FUNCTION_BLOCK Motor_VS (* CAT Function Block Type *)
  (* Standard: 61499-2 *)
  (* Version 0.0, 6/2/2026, Schneider Electric, template *)
  PACKAGE SE.Nereda;
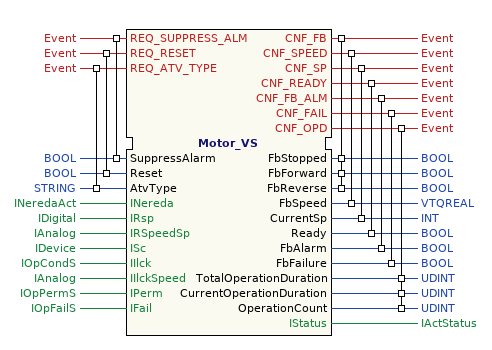
  EVENT_INPUT
    REQ_SUPPRESS_ALM WITH SuppressAlarm; (* Request to update the alarm suppress status *)
    REQ_RESET WITH Reset; (* Request to reset the device *)
    REQ_ATV_TYPE WITH AtvType;
  END_EVENT
  EVENT_OUTPUT
    CNF_FB WITH FbStopped, FbForward, FbReverse; (* Execution of confirmed state *)
    CNF_SPEED WITH FbSpeed; (* Execution of confirmed state *)
    CNF_SP WITH CurrentSp; (* Execution of confirmation current setpoint *)
    CNF_READY WITH Ready; (* Execution of Ready status *)
    CNF_FB_ALM WITH FbAlarm; (* Execution of confirmation  Fb alarm *)
    CNF_FAIL WITH FbFailure; (* Execution of confirmation  failure *)
    CNF_OPD WITH TotalOperationDuration, CurrentOperationDuration, OperationCount; (* Execution confirmation of operation durations *)
  END_EVENT
  VAR_INPUT
    SuppressAlarm : BOOL; (* 1 = Suppress alarm in HMI *)
    Reset : BOOL; (* 1 = Reset device failure *)
    AtvType : STRING;
  END_VAR
  VAR_OUTPUT
    FbStopped : BOOL; (* 1 = Stopped *)
    FbForward : BOOL; (* 1 = Running *)
    FbReverse : BOOL; (* 1 = Running *)
    FbSpeed : VTQREAL; (* Value from the hardware module *)
    CurrentSp : INT; (* Current output value considering permissive conditions *)
    Ready : BOOL; (* 1 = Device is ready to run *)
    FbAlarm : BOOL; (* 1 = Feedback failure alarm is active *)
    FbFailure : BOOL; (* 1 = Fail active *)
    TotalOperationDuration : UDINT; (* Total operation duration in minutes *)
    CurrentOperationDuration : UDINT; (* Current operational duration in minutes *)
    OperationCount : UDINT; (* Total operations count *)
  END_VAR
  SOCKETS
    INereda : INeredaAct;
  END_SOCKETS
  SOCKETS
    IRsp : IDigital; (* Program remote setpoint interface adapter *)
    IRSpeedSp : IAnalog; (* Program remote speed setpoint interface adpter, Controls the block when owner is in program local. *)
    ISc : IDevice; (* Sequence control Interface adapter. Controls the block when owner is in program local *)
    IIlck : IOpCondS; (* Condition summary chain input from upstream blocks *)
    IIlckSpeed : IAnalog; (* Speed setpoint to be considered if interlock condition is active *)
    IPerm : IOpPermS; (* Permission condition summary chain input from permCondItem blocks *)
    IFail : IOpFailS; (* Fail condition summary chain input from failCondItem blocks *)
  END_SOCKETS
  PLUGS
    IStatus : IActStatus;
  END_PLUGS
  (* 01 - FUNCTIONNAL INPUT INTERFACE *)
  (* 00 - INITIALIZATION *)
  (* 05 - LOGIC *)
  (* 06 - HMI INTERFACE *)
  (* 04 - CHILDREN *)
  (* 03 - FIELD INTERFACE *)
  (* 02 - FUNCTIONNAL OUTPUT INTERFACE *)
  (* 07- Input Hardware Interface *)
  (* 08- Output Hardware Interface *)
  (* 09- Local Panel *)
  (* Maintenance *)
  (* Fb Stop *)
  (* Interlock *)
  (* Mode *)
  (* Permissive *)
  (* 4A - TYPICALS *)
  (* Craeted By Nouriddin OUECHEN *)
  (* Failure *)
  (* Sequence Control *)
  (* Service Connection *)
  (* Reset *)
  (* FbRunning *)
  (* SetPoint *)
  (* Simulation (To be Removed) *)
  (* 07- ±OTOR VS ALARM *)
  (* Comment When `SafetySwitchOff = TRUE`, it means that the safety switch is **OFF**. *)
  FBS
    IThis : Motor_VS_HMI(QI := TRUE);
    INIT : plcStart(Prio := 35, Delay := T#0ms);
    extControlled : dISignal(Name := '$${PATH}DIn'); {SET_ATTRIBUTE(Configuration.Component.HideUnusedPorts, )}
    LocalPanel : FieldSignals;
    maintenance : DevMnt; {SET_ATTRIBUTE(Configuration.Component.HideUnusedPorts, )}
    NotRevFwd : NOT_425622A9A4AC6C60; {SET_ATTRIBUTE(Configuration.GenericFBType.InterfaceParams, Runtime.Standard#CNT:=2;OUT${CNT$}:BOOL,BOOL)}
    interlock : IlckCondSum; {SET_ATTRIBUTE(Configuration.Component.HideUnusedPorts, )}
    failure : FailCondSum; {SET_ATTRIBUTE(Configuration.Component.HideUnusedPorts, )}
    DriveFailure : failCondItem(CondCause := Active1); {SET_ATTRIBUTE(Configuration.Component.HideUnusedPorts, )}
    AtvFailure : SELECT_81F91C08E00C8B28(IN1 := FALSE); {SET_ATTRIBUTE(Configuration.GenericFBType.InterfaceParams, Runtime.Standard#CNT:=2;SELECT:BOOL;IN${CNT$}:BOOL)}
    ElectricCircuitFailure : failCondItem(CondCause := Active1); {SET_ATTRIBUTE(Configuration.Component.HideUnusedPorts, )}
    FrequencyInverterFailure : failCondItem(CondCause := Active1); {SET_ATTRIBUTE(Configuration.Component.HideUnusedPorts, )}
    PowerFailure : failCondItem(CondCause := Active1); {SET_ATTRIBUTE(Configuration.Component.HideUnusedPorts, )}
    CurrOwner : CurrOwnerDecode;
    State : ActState(pin_DD241BABAE81E6FD := Motor);
    NoPowerFb : NOT_42C76073DCEB1A7A; {SET_ATTRIBUTE(Configuration.GenericFBType.InterfaceParams, Runtime.Standard#CNT:=1;OUT${CNT$}:BOOL)}
    permissive : PermCondSum; {SET_ATTRIBUTE(Configuration.Component.HideUnusedPorts, )}
    BaseVs : MotorVsBase;
    interlockMotVs : IlckMotVs;
    fbFwd : dISignal(Name := '$${PATH}DIn'); {SET_ATTRIBUTE(Configuration.Component.HideUnusedPorts, )}
    fbRev : dISignal(Name := '$${PATH}DIn'); {SET_ATTRIBUTE(Configuration.Component.HideUnusedPorts, )}
    fbSpeed : aISignal(Name := '$${PATH}AIn'); (* (Minimum Value  = 0.0, Maximum Value = 100.0) *) {SET_ATTRIBUTE(Configuration.Component.HideUnusedPorts, )}
    FbStop : AND_88A3DD8EC65DD11C; {SET_ATTRIBUTE(Configuration.GenericFBType.InterfaceParams, Runtime.Standard#CNT:=2;OUT:BOOL)}
    serviceManager : MotorVsServiceManager; {SET_ATTRIBUTE(Configuration.Component.HideUnusedPorts, )}
    cmdFwd : dOSignal(Name := '$${PATH}DOut'); {SET_ATTRIBUTE(Configuration.Component.HideUnusedPorts, )}
    cmdSpeed : aOSignal(Name := '$${PATH}AOut'); {SET_ATTRIBUTE(Configuration.Component.HideUnusedPorts, )}
    cmdRev : dOSignal(Name := '$${PATH}DOut'); {SET_ATTRIBUTE(Configuration.Component.HideUnusedPorts, )}
    ResetCmd : OR_169B00D031196E7C4; {SET_ATTRIBUTE(Configuration.GenericFBType.InterfaceParams, Runtime.Standard#CNT:=4;OUT:BOOL)}
    FbRunning : OR_88A3DD8EC65DD11C; {SET_ATTRIBUTE(Configuration.GenericFBType.InterfaceParams, Runtime.Standard#CNT:=2;OUT:BOOL)}
    ISc1ISc2 : mergeIDevice;
    Sp : IDeviceEncode;
    IScISeqData : IScISecData;
    TRIP : failCondItem(CondCause := Active1); {SET_ATTRIBUTE(Configuration.Component.HideUnusedPorts, )}
    MoistureDetectionPumpMS : failCondItem(CondCause := Active1); {SET_ATTRIBUTE(Configuration.Component.HideUnusedPorts, )}
    Reset_Init : DS_SELECTX_2536758B411A6CE51(DI1_1 := TRUE, DI2_1 := FALSE); {SET_ATTRIBUTE(Configuration.GenericFBType.InterfaceParams, Runtime.Standard#CNTX:=2;CNTY:=1;DI${CNTX,_,CNTY$}:BOOL)}
    NoNeedReset : E_PERMIT;
    NotNeedReset : NOT_42C76073DCEB1A7A; {SET_ATTRIBUTE(Configuration.GenericFBType.InterfaceParams, Runtime.Standard#CNT:=1;OUT${CNT$}:BOOL)}
    SpeedSp : SpeedSp;
    SafetySwitchOff : ilckCondItem(CondCause := Active1);
    SafetySwitch : NOT_42C76073DCEB1A7A; {SET_ATTRIBUTE(Configuration.GenericFBType.InterfaceParams, Runtime.Standard#CNT:=1;OUT${CNT$}:BOOL)}
    AllFailures : OR_1147623A96AA66A8; {SET_ATTRIBUTE(Configuration.GenericFBType.InterfaceParams, Runtime.Standard#CNT:=7;OUT:BOOL)}
    AlarmDriveFailure : ALARM_BIT(ACKTYPE_1 := 2, ACTIVE := TRUE, TYPE := 1);
    AlarmTRIP : ALARM_BIT(ACKTYPE_1 := 2, TYPE := 1, ACTIVE := TRUE);
    AlarmElectricCircuitFailure : ALARM_BIT(ACKTYPE_1 := 2, ACTIVE := TRUE, TYPE := 1);
    AlarmFrequencyInverterFailure : ALARM_BIT(ACKTYPE_1 := 2, ACTIVE := TRUE, TYPE := 1);
    AlarmPowerFailure : ALARM_BIT(ACKTYPE_1 := 2, ACTIVE := TRUE, TYPE := 1);
    AlarmMoistureDetectionPumpMS : ALARM_BIT(ACKTYPE_1 := 2, ACTIVE := TRUE, TYPE := 1);
    MotorVsFailuresAlarms : MotVsFailures;
    MUL1 : MUL_1329C2AB45109BAAB(IN2 := 0.6); {SET_ATTRIBUTE(Configuration.GenericFBType.InterfaceParams, Runtime.Standard#CNT:=2;IN${CNT$}:REAL)}
    SYMLINKMULTIVARSRC1 : SYMLINKMULTIVARSRC_5A03F112CD5D470(QI := TRUE, NAME1 := '$${PATH}cmdFrequency'); {SET_ATTRIBUTE(Configuration.GenericFBType.InterfaceParams, Runtime.System#I:=1;VALUE${I$}:INT)}
    REAL2INT1 : REAL2INT;
    SYMLINKMULTIVARSRC2 : SYMLINKMULTIVARSRC_5A03F112CD5D470(QI := TRUE, NAME1 := '$${PATH}cmdSpeedINT'); {SET_ATTRIBUTE(Configuration.GenericFBType.InterfaceParams, Runtime.System#I:=1;VALUE${I$}:INT)}
    SpeedRawOut : speedToRawInt(pin_EEBD45F5182DE80D := 100.0);
    FbSpeedAdapter : speedFbAdapter(pin_919EBDC14EE69C57 := 100.0);
    fbSpeedINT : SYMLINKMULTIVARDST_5A03F112CD5D470(QI := TRUE, NAME1 := '$${PATH}fbSpeedINT'); {SET_ATTRIBUTE(Configuration.GenericFBType.InterfaceParams, Runtime.System#I:=1;VALUE${I$}:INT)}
  END_FBS
  EVENT_CONNECTIONS
    extControlled.CNF TO BaseVs.REQ_EXT_CTL;
    failure.COND_IND TO BaseVs.REQ_FAIL;
    REQ_SUPPRESS_ALM TO BaseVs.REQ_SUPPRESS_ALM;
    BaseVs.CNF_FB_STS TO CNF_FB;
    BaseVs.CNF_FB_ALM TO CNF_FB_ALM;
    State.7E9F7DF9BBDC513D TO CNF_FAIL;
    NoPowerFb.CNF TO DriveFailure.REQ;
    NoPowerFb.CNF TO ElectricCircuitFailure.REQ;
    NoPowerFb.CNF TO FrequencyInverterFailure.REQ;
    NoPowerFb.CNF TO PowerFailure.REQ;
    permissive.PERM_IND TO BaseVs.REQ_PERM;
    AtvFailure.CNF TO NoPowerFb.REQ;
    FbSpeedAdapter.DCDCAD18DFD61DDE TO BaseVs.REQ_FB_SPEED;
    fbFwd.CNF TO NotRevFwd.REQ;
    fbRev.CNF TO NotRevFwd.REQ;
    FbStop.CNF TO BaseVs.REQ_FB;
    NotRevFwd.CNF TO FbStop.REQ;
    BaseVs.CNF_OUT TO cmdFwd.REQ;
    BaseVs.CNF_OUT TO cmdRev.REQ;
    BaseVs.CNF_SPEED_OUT TO cmdSpeed.REQ;
    FbSpeedAdapter.DCDCAD18DFD61DDE TO CNF_SPEED;
    BaseVs.CNF_SP TO CNF_SP;
    maintenance.CNF_OPD TO CNF_OPD;
    BaseVs.CNF_FB_STS TO FbRunning.REQ;
    NoPowerFb.CNF TO TRIP.REQ;
    NoPowerFb.CNF TO MoistureDetectionPumpMS.REQ;
    REQ_RESET TO ResetCmd.REQ;
    ResetCmd.CNF TO BaseVs.REQ_RESET;
    Reset_Init.IND TO ResetCmd.REQ;
    NotNeedReset.CNF TO NoNeedReset.EI;
    BaseVs.CNF_NEED_RESET TO NotNeedReset.REQ;
    NoNeedReset.EO TO Reset_Init.REQ2;
    LocalPanel.08EBB16DA2AE2E53 TO AtvFailure.REQ;
    CurrOwner.7B1DE71047870DF3 TO State.503DFB34A9D9F842;
    State.B9B326A02DDC85D5 TO AlarmDriveFailure.INIT;
    State.B9B326A02DDC85D5 TO NotRevFwd.REQ;
    State.B9B326A02DDC85D5 TO IScISeqData.68E777F8FBF99C3F;
    State.B9B326A02DDC85D5 TO Sp.6454C45AB89C818D;
    State.B9B326A02DDC85D5 TO Reset_Init.REQ1;
    State.3E2F994B40CA5D8A TO CNF_READY;
    State.3E2F994B40CA5D8A TO INereda.CC753684FA882790;
    State.3E2F994B40CA5D8A TO IStatus.14377629A1F197A9;
    REQ_ATV_TYPE TO LocalPanel.62FE49324B71C4B0;
    FbRunning.CNF TO INereda.9CD053F8408797ED;
    FbSpeedAdapter.DCDCAD18DFD61DDE TO INereda.F846995A4121D865;
    BaseVs.CNF_FB_ALM TO INereda.C79FD2A34D0395C5;
    State.7E9F7DF9BBDC513D TO INereda.476AAA40EB7AA926;
    maintenance.CNF_OPD TO INereda.2DA8AEC15204E92D;
    INereda.0F1CDF9A9B4A227A TO BaseVs.REQ_SP;
    INereda.0F1CDF9A9B4A227A TO Sp.7A6C1C05B7ACA4D3;
    INereda.0F1CDF9A9B4A227A TO SpeedSp.3B62B1C54EE8482F;
    INereda.1E00729184986247 TO SpeedSp.3B62B1C54EE8482F;
    INereda.37BBC1F841739733 TO Sp.8DD7A09A6565B7F3;
    INereda.37BBC1F841739733 TO ResetCmd.REQ;
    SpeedSp.CE921AF394A1453E TO Sp.51FC99EF6C596181;
    BaseVs.CNF_MODE TO interlockMotVs.BB07CE5CA3A90E8C;
    BaseVs.CNF_OWNER TO interlockMotVs.47593EB5799F5830;
    interlockMotVs.1ACB26BE744F37A1 TO BaseVs.REQ_ILCK;
    FbRunning.CNF TO IStatus.14377629A1F197A9;
    FbSpeedAdapter.DCDCAD18DFD61DDE TO IStatus.03F1F1C982EE8DD5;
    SafetySwitch.CNF TO SafetySwitchOff.REQ;
    LocalPanel.08EBB16DA2AE2E53 TO SafetySwitch.REQ;
    LocalPanel.08EBB16DA2AE2E53 TO AllFailures.REQ;
    BaseVs.CNF_SP TO AllFailures.REQ;
    BaseVs.CNF_FB_STS TO AllFailures.REQ;
    BaseVs.CNF_OWNER TO AllFailures.REQ;
    BaseVs.CNF_READY TO AllFailures.REQ;
    BaseVs.CNF_MODE TO AllFailures.REQ;
    interlockMotVs.1ACB26BE744F37A1 TO AllFailures.REQ;
    BaseVs.CNF_FAIL TO AllFailures.REQ;
    AllFailures.CNF TO CurrOwner.3D8B91432EBB5812;
    NoPowerFb.CNF TO AllFailures.REQ;
    BaseVs.CNF_NEED_RESET TO AllFailures.REQ;
    AlarmPowerFailure.INITO TO AlarmTRIP.INIT;
    AlarmDriveFailure.INITO TO AlarmElectricCircuitFailure.INIT;
    AlarmElectricCircuitFailure.INITO TO AlarmFrequencyInverterFailure.INIT;
    AlarmDriveFailure.CNF_INITDATA TO AlarmDriveFailure.REQ;
    MotorVsFailuresAlarms.C14C3E40270A0244 TO AlarmDriveFailure.REQ_INITDATA;
    MotorVsFailuresAlarms.C14C3E40270A0244 TO AlarmTRIP.REQ_INITDATA;
    AlarmTRIP.CNF_INITDATA TO AlarmTRIP.REQ;
    AlarmDriveFailure.CNF_INITDATA TO AlarmDriveFailure.ACTIVATE;
    AlarmTRIP.CNF_INITDATA TO AlarmTRIP.ACTIVATE;
    AlarmFrequencyInverterFailure.INITO TO AlarmPowerFailure.INIT;
    MotorVsFailuresAlarms.C14C3E40270A0244 TO AlarmElectricCircuitFailure.REQ_INITDATA;
    MotorVsFailuresAlarms.C14C3E40270A0244 TO AlarmFrequencyInverterFailure.REQ_INITDATA;
    MotorVsFailuresAlarms.C14C3E40270A0244 TO AlarmPowerFailure.REQ_INITDATA;
    AlarmElectricCircuitFailure.CNF_INITDATA TO AlarmElectricCircuitFailure.ACTIVATE;
    AlarmElectricCircuitFailure.CNF_INITDATA TO AlarmElectricCircuitFailure.REQ;
    AlarmFrequencyInverterFailure.CNF_INITDATA TO AlarmFrequencyInverterFailure.ACTIVATE;
    AlarmFrequencyInverterFailure.CNF_INITDATA TO AlarmFrequencyInverterFailure.REQ;
    AlarmPowerFailure.CNF_INITDATA TO AlarmPowerFailure.ACTIVATE;
    AlarmPowerFailure.CNF_INITDATA TO AlarmPowerFailure.REQ;
    MotorVsFailuresAlarms.C14C3E40270A0244 TO AlarmMoistureDetectionPumpMS.REQ_INITDATA;
    AlarmMoistureDetectionPumpMS.CNF_INITDATA TO AlarmMoistureDetectionPumpMS.ACTIVATE;
    AlarmMoistureDetectionPumpMS.CNF_INITDATA TO AlarmMoistureDetectionPumpMS.REQ;
    AlarmTRIP.INITO TO AlarmMoistureDetectionPumpMS.INIT;
    NoPowerFb.CNF TO AlarmDriveFailure.REQ;
    NoPowerFb.CNF TO AlarmElectricCircuitFailure.REQ;
    NoPowerFb.CNF TO AlarmFrequencyInverterFailure.REQ;
    NoPowerFb.CNF TO AlarmPowerFailure.REQ;
    NoPowerFb.CNF TO AlarmTRIP.REQ;
    NoPowerFb.CNF TO AlarmMoistureDetectionPumpMS.REQ;
    AlarmMoistureDetectionPumpMS.INITO TO MotorVsFailuresAlarms.5D68F3F24BC03060;
    AlarmDriveFailure.IND_1 TO MotorVsFailuresAlarms.BB7D0193D5CDB632;
    AlarmElectricCircuitFailure.IND_1 TO MotorVsFailuresAlarms.BB7D0193D5CDB632;
    AlarmFrequencyInverterFailure.IND_1 TO MotorVsFailuresAlarms.BB7D0193D5CDB632;
    AlarmPowerFailure.IND_1 TO MotorVsFailuresAlarms.BB7D0193D5CDB632;
    AlarmTRIP.IND_1 TO MotorVsFailuresAlarms.BB7D0193D5CDB632;
    AlarmMoistureDetectionPumpMS.IND_1 TO MotorVsFailuresAlarms.BB7D0193D5CDB632;
    INIT.FIRST_INIT TO IThis.5D65C7F23F6CCFDB;
    INIT.REDO_INIT TO IThis.5D65C7F23F6CCFDB;
    State.B9B326A02DDC85D5 TO IThis.D29F1FADF6E57358;
    LocalPanel.08EBB16DA2AE2E53 TO IThis.438D25703EEFF814;
    BaseVs.CNF_SPEED_SP TO IThis.0316FFC0BDC899BE;
    FbSpeedAdapter.DCDCAD18DFD61DDE TO IThis.0316FFC0BDC899BE;
    BaseVs.CNF_NEED_RESET TO IThis.05E2BC0E0C273F8B;
    State.7E9F7DF9BBDC513D TO IThis.A2D93536FF9B406B;
    fbFwd.CNF TO IThis.C9F8920D38B4A811;
    IThis.141F2765F0199247 TO State.747A80A26976E9BA;
    IThis.EDABC861E1C71398 TO AtvFailure.REQ;
    IThis.6535878B6880E95C TO ResetCmd.REQ;
    IThis.52FEB725938026A3 TO BaseVs.REQ_SPEED_SP;
    BaseVs.CNF_SPEED_OUT TO MUL1.REQ;
    MUL1.CNF TO REAL2INT1.DD5870AA881150BB;
    MotorVsFailuresAlarms.C14C3E40270A0244 TO fbSpeedINT.INIT;
    REAL2INT1.6FC99A5BD1C38561 TO SYMLINKMULTIVARSRC1.REQ;
    SYMLINKMULTIVARSRC1.INITO TO INIT.ACK_FIRST;
    BaseVs.CNF_SPEED_OUT TO SpeedRawOut.45891852F5D66F4B;
    SpeedRawOut.73091BCABFCCFCB6 TO SYMLINKMULTIVARSRC2.REQ;
    SYMLINKMULTIVARSRC2.INITO TO SYMLINKMULTIVARSRC1.INIT;
    fbSpeed.CNF TO FbSpeedAdapter.23AEC014E6AA5B8A;
    fbSpeedINT.CNF TO FbSpeedAdapter.D15EB431906F2F27;
    fbSpeedINT.INITO TO SYMLINKMULTIVARSRC2.INIT;
  END_CONNECTIONS
  DATA_CONNECTIONS
    extControlled.Out TO BaseVs.ExternalControlled;
    fbFwd.Out TO BaseVs.FbFwd;
    failure.State TO BaseVs.Fail;
    SuppressAlarm TO BaseVs.SuppressAlarm;
    BaseVs.FbStopped TO FbStopped;
    BaseVs.FbFwdRunning TO FbForward;
    BaseVs.FbAlarm TO FbAlarm;
    State.8CCAFBE354ECA569 TO FbFailure;
    AtvFailure.OUT TO DriveFailure.CondSignal;
    NoPowerFb.OUT1 TO PowerFailure.CondSignal;
    permissive.PermPassive TO BaseVs.PermStop;
    permissive.PermActive1 TO BaseVs.PermFwd;
    fbRev.Out TO BaseVs.FbRev;
    FbSpeedAdapter.02242968B1987D9E TO BaseVs.FbSpeed;
    fbFwd.Out TO NotRevFwd.IN1;
    FbStop.OUT TO BaseVs.FbStop;
    fbRev.Out TO NotRevFwd.IN2;
    NotRevFwd.OUT1 TO FbStop.IN1;
    NotRevFwd.OUT2 TO FbStop.IN2;
    permissive.PermActive2 TO BaseVs.PermRev;
    BaseVs.OutFwd TO cmdFwd.Signal;
    BaseVs.OutRev TO cmdRev.Signal;
    BaseVs.OutSpeed TO cmdSpeed.Signal;
    FbSpeedAdapter.02242968B1987D9E TO FbSpeed;
    BaseVs.FbRevRunning TO FbReverse;
    BaseVs.CurrentSp TO CurrentSp;
    maintenance.TotalOperationDuration TO TotalOperationDuration;
    maintenance.CurrentOperationDuration TO CurrentOperationDuration;
    maintenance.OperationCount TO OperationCount;
    BaseVs.FbFwdRunning TO FbRunning.IN1;
    BaseVs.FbRevRunning TO FbRunning.IN2;
    Reset TO ResetCmd.IN1;
    ResetCmd.OUT TO BaseVs.Reset;
    Reset_Init.OUT1 TO ResetCmd.IN4;
    NotNeedReset.OUT1 TO NoNeedReset.PERMIT;
    BaseVs.NeedReset TO NotNeedReset.IN1;
    LocalPanel.9DA3D6735086B77A TO ElectricCircuitFailure.CondSignal;
    LocalPanel.B021B183D08305E2 TO FrequencyInverterFailure.CondSignal;
    LocalPanel.DA445F1C2864A153 TO State.C70237F918BB93F6;
    LocalPanel.B46B24B64003C584 TO NoPowerFb.IN1;
    LocalPanel.B46B24B64003C584 TO State.655DE7D6E2CF8FB8;
    LocalPanel.61B515FEF739774D TO AtvFailure.IN2;
    LocalPanel.4379EE93CED9D91D TO TRIP.CondSignal;
    LocalPanel.5EFEAD483C25BA7B TO MoistureDetectionPumpMS.CondSignal;
    CurrOwner.CEBE936F1EA616DB TO State.E90E39DE4A80ABDE;
    CurrOwner.1FF13EB8D921FC26 TO State.3885B231A80F7FFF;
    BaseVs.CurrentOwner TO CurrOwner.B2DAC483AB345195;
    State.4E509FA35DBACB85 TO Ready;
    State.4E509FA35DBACB85 TO INereda.8A8A07EFCDA1443C;
    State.4E509FA35DBACB85 TO IStatus.9E0B44559326BEAF;
    BaseVs.CurrentSp TO State.52C3EF6D9E750127;
    BaseVs.FbStatus TO State.8E076A9FED13120E;
    BaseVs.Ready TO State.1C9201C719ABF50B;
    BaseVs.Simulation TO State.7A0BDA68B634A263;
    BaseVs.FbOverride TO State.DD66F5DCF7F6FB1D;
    interlockMotVs.74F62D32B8AB17CB TO State.9A204E382C1350DC;
    AtvType TO LocalPanel.62A70FF94078EC4D;
    BaseVs.FbStopped TO INereda.D83B5BDEFA4D797C;
    FbRunning.OUT TO INereda.B762734C094A7162;
    BaseVs.FbFwdRunning TO INereda.13E1B1B6EE0F07DB;
    BaseVs.FbRevRunning TO INereda.3011FF733C667A56;
    FbSpeedAdapter.02242968B1987D9E TO INereda.790C5C3BA88E0AF5;
    BaseVs.FbAlarm TO INereda.BDD69968F2D82EAF;
    State.8CCAFBE354ECA569 TO INereda.6EEAF63EEE6021B6;
    maintenance.TotalOperationDuration TO INereda.C7F638DBF6B860D2;
    maintenance.CurrentOperationDuration TO INereda.9224E22E0E82A2D7;
    maintenance.OperationCount TO INereda.10624535249F94F3;
    INereda.710D7FC54EE3F35A TO BaseVs.Sp;
    INereda.710D7FC54EE3F35A TO Sp.64F0A65D5B10944D;
    INereda.710D7FC54EE3F35A TO SpeedSp.28B1E385E2B35AAE;
    INereda.1BC103921BBFDA0B TO SpeedSp.79740CC6CE911CBD;
    INereda.EA28053F07575F36 TO Sp.48AF5FD15A286274;
    INereda.EA28053F07575F36 TO ResetCmd.IN3;
    SpeedSp.335EA17E377251F8 TO Sp.35DB549676DB86DA;
    BaseVs.Maintenance TO interlockMotVs.3100FF95313D2E79;
    BaseVs.CurrentOwner TO interlockMotVs.B24A2EB6CD7D5206;
    interlockMotVs.5B70B8A759686CBA TO BaseVs.IlckPos;
    interlockMotVs.5CCAAE9E9D3EC477 TO BaseVs.IlckType;
    interlockMotVs.7BFBF177262F6463 TO BaseVs.IlckSpeed;
    BaseVs.FbStopped TO IStatus.227987A2F0C6A825;
    FbRunning.OUT TO IStatus.D41A46B14EF7208D;
    FbSpeedAdapter.02242968B1987D9E TO IStatus.B9E42D72CEF16844;
    SafetySwitch.OUT1 TO SafetySwitchOff.CondSignal;
    LocalPanel.9F4FA80000721942 TO SafetySwitch.IN1;
    interlockMotVs.74F62D32B8AB17CB TO BaseVs.IlckCond;
    BaseVs.FbAlarm TO State.F37ACDE435F84908;
    BaseVs.FailStatus TO AllFailures.IN1;
    AtvFailure.OUT TO AllFailures.IN2;
    LocalPanel.9DA3D6735086B77A TO AllFailures.IN3;
    LocalPanel.B021B183D08305E2 TO AllFailures.IN4;
    NoPowerFb.OUT1 TO AllFailures.IN5;
    LocalPanel.4379EE93CED9D91D TO AllFailures.IN6;
    LocalPanel.5EFEAD483C25BA7B TO AllFailures.IN7;
    AllFailures.OUT TO State.94E3C396E1CCD1C0;
    BaseVs.NeedReset TO State.3ED730632EF45559;
    AtvFailure.OUT TO AlarmDriveFailure.INP;
    LocalPanel.9DA3D6735086B77A TO AlarmElectricCircuitFailure.INP;
    LocalPanel.B021B183D08305E2 TO AlarmFrequencyInverterFailure.INP;
    NoPowerFb.OUT1 TO AlarmPowerFailure.INP;
    LocalPanel.4379EE93CED9D91D TO AlarmTRIP.INP;
    LocalPanel.5EFEAD483C25BA7B TO AlarmMoistureDetectionPumpMS.INP;
    AlarmDriveFailure.STATE_1 TO MotorVsFailuresAlarms.CF590858835199A8;
    AlarmElectricCircuitFailure.STATE_1 TO MotorVsFailuresAlarms.E95D89BBD9B84237;
    AlarmFrequencyInverterFailure.STATE_1 TO MotorVsFailuresAlarms.9CDEFF528B20B5BB;
    AlarmPowerFailure.STATE_1 TO MotorVsFailuresAlarms.1283E3BFEB4BF28A;
    AlarmTRIP.STATE_1 TO MotorVsFailuresAlarms.1C3CFF04A8261C1D;
    AlarmMoistureDetectionPumpMS.STATE_1 TO MotorVsFailuresAlarms.ADEAB09FE145CE62;
    AlarmDriveFailure.COUNT_1 TO MotorVsFailuresAlarms.967C39787E15B333;
    AlarmElectricCircuitFailure.COUNT_1 TO MotorVsFailuresAlarms.3A0D63292928B9AE;
    AlarmFrequencyInverterFailure.COUNT_1 TO MotorVsFailuresAlarms.308E23D6E2FFA65B;
    AlarmPowerFailure.COUNT_1 TO MotorVsFailuresAlarms.B894C163AE8063C2;
    AlarmTRIP.COUNT_1 TO MotorVsFailuresAlarms.1FBA7DE6E18CD10B;
    AlarmMoistureDetectionPumpMS.COUNT_1 TO MotorVsFailuresAlarms.1CF94679776431BE;
    LocalPanel.9DA3D6735086B77A TO IThis.0AE962625433D46C;
    LocalPanel.61B515FEF739774D TO IThis.05CEFE840775FD43;
    BaseVs.CurrentSpeedSp TO IThis.0AC50FCC07E6318B;
    FbSpeedAdapter.02242968B1987D9E TO IThis.AE0C863666AF4242;
    BaseVs.NeedReset TO IThis.6B1BF7DB6EBC72CB;
    State.8CCAFBE354ECA569 TO IThis.E927219C5010AF15;
    fbFwd.Out TO IThis.1A624A669739224B;
    IThis.E887C120F3A4AF42 TO AtvFailure.SELECT;
    IThis.3B77DD9B964F7734 TO ResetCmd.IN2;
    IThis.3BD5B20D44F79E70 TO BaseVs.SpeedSpMin;
    IThis.5B58431AE2CD76E4 TO BaseVs.SpeedSpMax;
    BaseVs.OutSpeed TO MUL1.IN1;
    MUL1.OUT TO REAL2INT1.4573FC8F228EB71D;
    REAL2INT1.A6DEF5F9C27C1848 TO SYMLINKMULTIVARSRC1.VALUE1;
    BaseVs.OutSpeed TO SpeedRawOut.B2FF8AC2A57695C6;
    SpeedRawOut.0BBC678D1288C222 TO SYMLINKMULTIVARSRC2.VALUE1;
    fbSpeed.Out TO FbSpeedAdapter.18FE2B2470AA3359;
    fbSpeedINT.VALUE1 TO FbSpeedAdapter.A530287FDB8697A7;
    fbSpeedINT.QO TO FbSpeedAdapter.46C4F82F6CC69CD7;
  END_CONNECTIONS
  ADAPTER_CONNECTIONS
    IIlck TO SafetySwitchOff.ICondChainIn;
    IFail TO DriveFailure.ICondChainIn;
    DriveFailure.ICondChainOut TO ElectricCircuitFailure.ICondChainIn;
    ElectricCircuitFailure.ICondChainOut TO FrequencyInverterFailure.ICondChainIn;
    FrequencyInverterFailure.ICondChainOut TO PowerFailure.ICondChainIn;
    MoistureDetectionPumpMS.ICondChainOut TO failure.IOpCondIn;
    IPerm TO permissive.IOpPermIn;
    maintenance.IMaintenance TO serviceManager.IMaint;
    IRsp TO serviceManager.IRsp;
    IRSpeedSp TO serviceManager.IRSpeedSp;
    ISc TO ISc1ISc2.1;
    serviceManager.14 TO BaseVs.IServiceExtension;
    TRIP.ICondChainOut TO MoistureDetectionPumpMS.ICondChainIn;
    PowerFailure.ICondChainOut TO TRIP.ICondChainIn;
    ISc1ISc2.ISc TO IScISeqData.402225FF97C7FA69;
    Sp.3CE9C36DE62AE8E7 TO ISc1ISc2.2;
    IScISeqData.897A325283B7FA64 TO serviceManager.ISc;
    interlock.36 TO interlockMotVs.67B6C8BC3D21E047;
    IIlckSpeed TO interlockMotVs.8B394DC08166B07A;
    SafetySwitchOff.ICondChainOut TO interlock.IOpCondIn;
  END_CONNECTIONS
END_FUNCTION_BLOCK
